# EPICS substitutions: subTestApp/Db/user.substitutions
# Example substitutions file

file "db/circle.db" {
    { user = "bchandler" }
}

file "db/dbExample1.db" {
    { user = "bchandler" }
}

file db/dbExample2.db {
    pattern { user, no, scan }
        { "bchandler", 1, "1 second" }
        { "bchandler", 2, "2 second" }
        { "bchandler", 3, "5 second" }
}
